// TIA Portal V18 program export: 1 tag tables, 0 data types, 3 data blocks, 8 code blocks (in call order from the OBs), 5 instance data blocks

VAR_GLOBAL   // PLC tag table "Default tag table"
   Tag_1 AT %M0.0 : Bool;
   System_Byte AT %MB1 : Byte;
   FirstScan AT %M1.0 : Bool;
   DiagStatusUpdate AT %M1.1 : Bool;
   AlwaysTRUE AT %M1.2 : Bool;
   AlwaysFALSE AT %M1.3 : Bool;
   Clock_Byte AT %MB0 : Byte;
   Clock_10Hz AT %M0.0 : Bool;
   Clock_5Hz AT %M0.1 : Bool;
   "Clock_2.5Hz" AT %M0.2 : Bool;
   Clock_2Hz AT %M0.3 : Bool;
   "Clock_1.25Hz" AT %M0.4 : Bool;
   Clock_1Hz AT %M0.5 : Bool;
   "Clock_0.625Hz" AT %M0.6 : Bool;
   "Clock_0.5Hz" AT %M0.7 : Bool;
   Tag_2 AT %M10.0 : Bool;
   Tag_3 AT %MW20 : Word;
   Tag_4 AT %M20.1 : Bool;
   Tag_5 AT %MD20 : Real;
   Tag_6 AT %M10.7 : Bool;
   Tag_7 AT %MD30 : DWord;
   Tag_8 AT %M10.5 : Bool;
END_VAR

DATA_BLOCK "DATA"   // DB2
{ S7_Optimized_Access := 'TRUE' }
VERSION : 0.1
// stored: AutoNumber true, DBAccessibleFromOPCUA true, DBAccessibleFromWebserver true, IsOnlyStoredInLoadMemory false, IsRetainMemResEnabled false, IsWriteProtectedInAS false, MemoryReserve 100
   VAR
      Str : String := '0+252+65526+5000+955+54+100+566';
      Str_1 : String[4];
      Val_1 : DInt;
      Val_2 : DInt;
      Val_3 : DInt;
   END_VAR
BEGIN
END_DATA_BLOCK

DATA_BLOCK "DB_CLOUD"   // DB1201
{ S7_Optimized_Access := 'FALSE' }
VERSION : 0.1
// stored: AutoNumber false, DBAccessibleFromOPCUA true, DBAccessibleFromWebserver true, IsOnlyStoredInLoadMemory false, IsWriteProtectedInAS false
   VAR
      P1S1O2 : Real := 1.0;
      P1S1CO2 : Real := 2.0;
      P1S1MT : Real := 3.0;
      P1S1H : Real := 4.0;
      P1S1PH : Real := 5.0;
      P1S2O2 : Real := 1.0;
      P1S2CO2 : Real := 2.0;
      P1S2MT : Real := 3.0;
      P1S2H : Real := 4.0;
      P1S2PH : Real := 5.0;
      P1S3O2 : Real := 1.0;
      P1S3CO2 : Real := 2.0;
      P1S3MT : Real := 3.0;
      P1S3H : Real := 4.0;
      P1S3PH : Real := 5.0;
      P2S1O2 : Real := 1.0;
      P2S1CO2 : Real := 2.0;
      P2S1MT : Real := 3.0;
      P2S1H : Real := 4.0;
      P2S1PH : Real := 5.0;
      P2S2O2 : Real := 1.0;
      P2S2CO2 : Real := 2.0;
      P2S2MT : Real := 3.0;
      P2S2H : Real := 4.0;
      P2S2PH : Real := 5.0;
      P2S3O2 : Real := 1.0;
      P2S3CO2 : Real := 2.0;
      P2S3MT : Real := 3.0;
      P2S3H : Real := 4.0;
      P2S3PH : Real := 5.0;
      P3S1O2 : Real := 1.0;
      P3S1CO2 : Real := 2.0;
      P3S1MT : Real := 3.0;
      P3S1H : Real := 4.0;
      P3S1PH : Real := 5.0;
      P3S2O2 : Real := 1.0;
      P3S2CO2 : Real := 2.0;
      P3S2MT : Real := 3.0;
      P3S2H : Real := 4.0;
      P3S2PH : Real := 5.0;
      P3S3O2 : Real := 1.0;
      P3S3CO2 : Real := 2.0;
      P3S3MT : Real := 3.0;
      P3S3H : Real := 4.0;
      P3S3PH : Real := 5.0;
      P4S1O2 : Real := 1.0;
      P4S1CO2 : Real := 2.0;
      P4S1MT : Real := 3.0;
      P4S1H : Real := 4.0;
      P4S1PH : Real := 5.0;
      P4S2O2 : Real := 1.0;
      P4S2CO2 : Real := 2.0;
      P4S2MT : Real := 3.0;
      P4S2H : Real := 4.0;
      P4S2PH : Real := 5.0;
      P4S3O2 : Real := 1.0;
      P4S3CO2 : Real := 2.0;
      P4S3MT : Real := 3.0;
      P4S3H : Real := 4.0;
      P4S3PH : Real := 5.0;
      P5S1O2 : Real := 1.0;
      P5S1CO2 : Real := 2.0;
      P5S1MT : Real := 3.0;
      P5S1H : Real := 4.0;
      P5S1PH : Real := 5.0;
      P5S2O2 : Real := 1.0;
      P5S2CO2 : Real := 2.0;
      P5S2MT : Real := 3.0;
      P5S2H : Real := 4.0;
      P5S2PH : Real := 5.0;
      P5S3O2 : Real := 1.0;
      P5S3CO2 : Real := 2.0;
      P5S3MT : Real := 3.0;
      P5S3H : Real := 4.0;
      P5S3PH : Real := 5.0;
      P6S1O2 : Real := 1.0;
      P6S1CO2 : Real := 2.0;
      P6S1MT : Real := 3.0;
      P6S1H : Real := 4.0;
      P6S1PH : Real := 5.0;
      P6S2O2 : Real := 1.0;
      P6S2CO2 : Real := 2.0;
      P6S2MT : Real := 3.0;
      P6S2H : Real := 4.0;
      P6S2PH : Real := 5.0;
      P6S3O2 : Real := 1.0;
      P6S3CO2 : Real := 2.0;
      P6S3MT : Real := 3.0;
      P6S3H : Real := 4.0;
      P6S3PH : Real := 5.0;
   END_VAR
BEGIN
END_DATA_BLOCK

DATA_BLOCK "DB_CLOUD_Simulation"   // DB1200
{ S7_Optimized_Access := 'FALSE' }
VERSION : 0.1
// stored: AutoNumber false, DBAccessibleFromOPCUA true, DBAccessibleFromWebserver true, IsOnlyStoredInLoadMemory false, IsWriteProtectedInAS false
   VAR RETAIN
      Array_1 : Array[1..90] of Real;
      P1S1CO2 : Real := 0.0;
      P1S1MT : Real := 1.0;
      P1S1H : Real := 2.0;
      P1S1PH : Real := 3.0;
      P1S2O2 : Real := 4.0;
      P1S2CO2 : Real := 5.0;
      P1S2MT : Real := 6.0;
      P1S2H : Real := 7.0;
      P1S2PH : Real := 8.0;
      P1S3O2 : Real := 9.0;
      P1S3CO2 : Real := 10.0;
      P1S3MT : Real := 11.0;
      P1S3H : Real := 12.0;
      P1S3PH : Real := 13.0;
      P2S1O2 : Real := 14.0;
      P2S1CO2 : Real := 15.0;
      P2S1MT : Real := 16.0;
      P2S1H : Real := 17.0;
      P2S1PH : Real := 18.0;
      P2S2O2 : Real := 19.0;
      P2S2CO2 : Real := 20.0;
      P2S2MT : Real := 21.0;
      P2S2H : Real := 22.0;
      P2S2PH : Real := 23.0;
      P2S3O2 : Real := 24.0;
      P2S3CO2 : Real := 25.0;
      P2S3MT : Real := 26.0;
      P2S3H : Real := 27.0;
      P2S3PH : Real := 28.0;
      P3S1O2 : Real := 29.0;
      P3S1CO2 : Real := 30.0;
      P3S1MT : Real := 31.0;
      P3S1H : Real := 32.0;
      P3S1PH : Real := 33.0;
      P3S2O2 : Real := 34.0;
      P3S2CO2 : Real := 35.0;
      P3S2MT : Real := 36.0;
      P3S2H : Real := 37.0;
      P3S2PH : Real := 38.0;
      P3S3O2 : Real := 39.0;
      P3S3CO2 : Real := 40.0;
      P3S3MT : Real := 41.0;
      P3S3H : Real := 42.0;
      P3S3PH : Real := 43.0;
      P4S1O2 : Real := 44.0;
      P4S1CO2 : Real := 45.0;
      P4S1MT : Real := 46.0;
      P4S1H : Real := 47.0;
      P4S1PH : Real := 48.0;
      P4S2O2 : Real := 49.0;
      P4S2CO2 : Real := 50.0;
      P4S2MT : Real := 51.0;
      P4S2H : Real := 52.0;
      P4S2PH : Real := 53.0;
      P4S3O2 : Real := 54.0;
      P4S3CO2 : Real := 55.0;
      P4S3MT : Real := 56.0;
      P4S3H : Real := 57.0;
      P4S3PH : Real := 58.0;
      P5S1O2 : Real := 59.0;
      P5S1CO2 : Real := 60.0;
      P5S1MT : Real := 61.0;
      P5S1H : Real := 62.0;
      P5S1PH : Real := 63.0;
      P5S2O2 : Real := 64.0;
      P5S2CO2 : Real := 65.0;
      P5S2MT : Real := 66.0;
      P5S2H : Real := 67.0;
      P5S2PH : Real := 68.0;
      P5S3O2 : Real := 69.0;
      P5S3CO2 : Real := 70.0;
      P5S3MT : Real := 71.0;
      P5S3H : Real := 72.0;
      P5S3PH : Real := 73.0;
      P6S1O2 : Real := 74.0;
      P6S1CO2 : Real := 75.0;
      P6S1MT : Real := 76.0;
      P6S1H : Real := 77.0;
      P6S1PH : Real := 78.0;
      P6S2O2 : Real := 79.0;
      P6S2CO2 : Real := 80.0;
      P6S2MT : Real := 81.0;
      P6S2H : Real := 82.0;
      P6S2PH : Real := 83.0;
      P6S3O2 : Real := 84.0;
      P6S3CO2 : Real := 85.0;
      P6S3MT : Real := 86.0;
      P6S3H : Real := 87.0;
      P6S3PH : Real := 88.0;
   END_VAR
BEGIN
   Array_1[1] := 0.0;
   Array_1[2] := 1.0;
   Array_1[3] := 2.0;
   Array_1[4] := 3.0;
   Array_1[5] := 4.0;
   Array_1[6] := 5.0;
   Array_1[7] := 6.0;
   Array_1[8] := 7.0;
   Array_1[9] := 8.0;
   Array_1[10] := 9.0;
   Array_1[11] := 10.0;
   Array_1[12] := 11.0;
   Array_1[13] := 12.0;
   Array_1[14] := 13.0;
   Array_1[15] := 14.0;
   Array_1[16] := 15.0;
   Array_1[17] := 16.0;
   Array_1[18] := 17.0;
   Array_1[19] := 18.0;
   Array_1[20] := 19.0;
   Array_1[21] := 20.0;
   Array_1[22] := 21.0;
   Array_1[23] := 22.0;
   Array_1[24] := 23.0;
   Array_1[25] := 24.0;
   Array_1[26] := 25.0;
   Array_1[27] := 26.0;
   Array_1[28] := 27.0;
   Array_1[29] := 28.0;
   Array_1[30] := 29.0;
   Array_1[31] := 30.0;
   Array_1[32] := 31.0;
   Array_1[33] := 32.0;
   Array_1[34] := 33.0;
   Array_1[35] := 34.0;
   Array_1[36] := 35.0;
   Array_1[37] := 36.0;
   Array_1[38] := 37.0;
   Array_1[39] := 38.0;
   Array_1[40] := 39.0;
   Array_1[41] := 40.0;
   Array_1[42] := 41.0;
   Array_1[43] := 42.0;
   Array_1[44] := 43.0;
   Array_1[45] := 44.0;
   Array_1[46] := 45.0;
   Array_1[47] := 46.0;
   Array_1[48] := 47.0;
   Array_1[49] := 48.0;
   Array_1[50] := 49.0;
   Array_1[51] := 50.0;
   Array_1[52] := 51.0;
   Array_1[53] := 52.0;
   Array_1[54] := 53.0;
   Array_1[55] := 54.0;
   Array_1[56] := 55.0;
   Array_1[57] := 56.0;
   Array_1[58] := 57.0;
   Array_1[59] := 58.0;
   Array_1[60] := 59.0;
   Array_1[61] := 60.0;
   Array_1[62] := 61.0;
   Array_1[63] := 62.0;
   Array_1[64] := 63.0;
   Array_1[65] := 64.0;
   Array_1[66] := 65.0;
   Array_1[67] := 66.0;
   Array_1[68] := 67.0;
   Array_1[69] := 68.0;
   Array_1[70] := 69.0;
   Array_1[71] := 70.0;
   Array_1[72] := 71.0;
   Array_1[73] := 72.0;
   Array_1[74] := 73.0;
   Array_1[75] := 74.0;
   Array_1[76] := 75.0;
   Array_1[77] := 76.0;
   Array_1[78] := 77.0;
   Array_1[79] := 78.0;
   Array_1[80] := 79.0;
   Array_1[81] := 80.0;
   Array_1[82] := 81.0;
   Array_1[83] := 82.0;
   Array_1[84] := 83.0;
   Array_1[85] := 84.0;
   Array_1[86] := 85.0;
   Array_1[87] := 86.0;
   Array_1[88] := 87.0;
   Array_1[89] := 88.0;
   Array_1[90] := 89.0;
END_DATA_BLOCK

ORGANIZATION_BLOCK "Main"   // OB1, LAD, ProgramCycle
TITLE = "Main Program Sweep (Cycle)"
{ S7_Optimized_Access := 'TRUE' }
VERSION : 0.1
// stored: AutoNumber true, IsIECCheckEnabled false, SetENOAutomatically false
   VAR_INPUT
      Initial_Call : Bool;   // Initial call of this OB
      Remanence : Bool;   // =True, if remanent data are available
   END_VAR
BEGIN

REGION Network 1
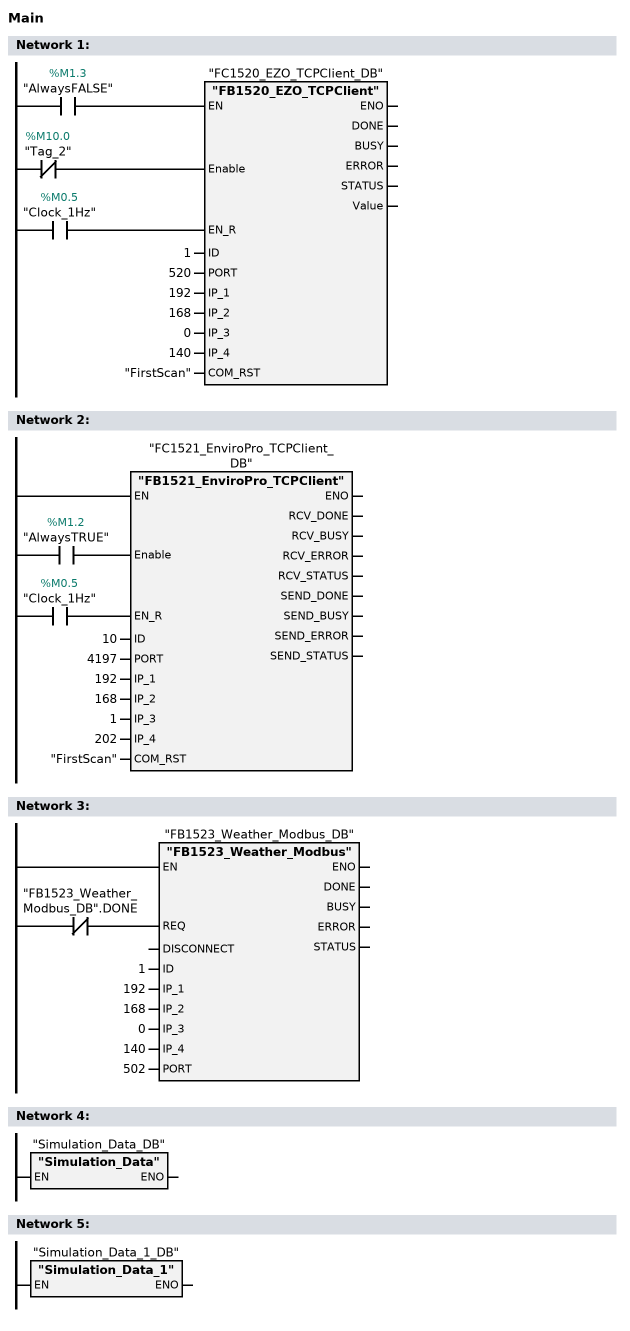
   RUNG wire#powerrail
      Contact( "AlwaysFALSE" )
      "FC1520_EZO_TCPClient_DB"(Enable := wire#w1, EN_R := wire#w2, ID := 1, PORT := 520, IP_1 := 192, IP_2 := 168, IP_3 := 0, IP_4 := 140, COM_RST := "FirstScan", DONE =>, BUSY =>, ERROR =>, STATUS =>, Value =>)
   END_RUNG
   RUNG wire#powerrail
      I_Contact( "Tag_2" )
   END_RUNG wire#w1
   RUNG wire#powerrail
      Contact( "Clock_1Hz" )
   END_RUNG wire#w2
   // the same network as SCL:
   IF "AlwaysFALSE" THEN
       "FC1520_EZO_TCPClient_DB"(Enable := NOT "Tag_2",   // "FB1520_EZO_TCPClient"
                               EN_R := "Clock_1Hz",
                               ID := 1,
                               PORT := 520,
                               IP_1 := 192,
                               IP_2 := 168,
                               IP_3 := 0,
                               IP_4 := 140,
                               COM_RST := "FirstScan");
   END_IF;
END_REGION

REGION Network 2
   RUNG wire#powerrail
      "FC1521_EnviroPro_TCPClient_DB"(Enable := wire#w1, EN_R := wire#w2, ID := 10, PORT := 4197, IP_1 := 192, IP_2 := 168, IP_3 := 1, IP_4 := 202, COM_RST := "FirstScan", RCV_DONE =>, RCV_BUSY =>, RCV_ERROR =>, RCV_STATUS =>, SEND_DONE =>, SEND_BUSY =>, SEND_ERROR =>, SEND_STATUS =>)
   END_RUNG
   RUNG wire#powerrail
      Contact( "AlwaysTRUE" )
   END_RUNG wire#w1
   RUNG wire#powerrail
      Contact( "Clock_1Hz" )
   END_RUNG wire#w2
   // the same network as SCL:
   "FC1521_EnviroPro_TCPClient_DB"(Enable := "AlwaysTRUE",   // "FB1521_EnviroPro_TCPClient"
                           EN_R := "Clock_1Hz",
                           ID := 10,
                           PORT := 4197,
                           IP_1 := 192,
                           IP_2 := 168,
                           IP_3 := 1,
                           IP_4 := 202,
                           COM_RST := "FirstScan");
END_REGION

REGION Network 3
   RUNG wire#powerrail
      "FB1523_Weather_Modbus_DB"(REQ := wire#w1, DISCONNECT :=, ID := 1, IP_1 := 192, IP_2 := 168, IP_3 := 0, IP_4 := 140, PORT := 502, DONE =>, BUSY =>, ERROR =>, STATUS =>)
   END_RUNG
   RUNG wire#powerrail
      I_Contact( "FB1523_Weather_Modbus_DB".DONE )
   END_RUNG wire#w1
   // the same network as SCL:
   "FB1523_Weather_Modbus_DB"(REQ := NOT "FB1523_Weather_Modbus_DB".DONE,   // "FB1523_Weather_Modbus"
                           ID := 1,
                           IP_1 := 192,
                           IP_2 := 168,
                           IP_3 := 0,
                           IP_4 := 140,
                           PORT := 502);
END_REGION

REGION Network 4
   RUNG wire#powerrail
      "Simulation_Data_DB"()
   END_RUNG
   // the same network as SCL:
   "Simulation_Data_DB"();   // "Simulation_Data"
END_REGION

REGION Network 5
   RUNG wire#powerrail
      "Simulation_Data_1_DB"()
   END_RUNG
   // the same network as SCL:
   "Simulation_Data_1_DB"();   // "Simulation_Data_1"
END_REGION
END_ORGANIZATION_BLOCK

FUNCTION_BLOCK "FB1520_EZO_TCPClient"
{ S7_Optimized_Access := 'TRUE' }
VERSION : 0.1
   VAR_INPUT 
      Enable : Bool;
      EN_R : Bool;
      ID : CONN_OUC := 16#0001;
      PORT : UInt := 4196;
      IP_1 : Byte := 192;
      IP_2 : Byte := 168;
      IP_3 : Byte := 1;
      IP_4 : Byte := 200;
   END_VAR

   VAR_OUTPUT 
      DONE : Bool;
      BUSY : Bool;
      ERROR : Bool;
      STATUS : Word;
      Value : Real;
   END_VAR

   VAR_IN_OUT 
      COM_RST : Bool;
   END_VAR

   VAR 
      CONNECT {InstructionName := 'TCON_IP_v4'; LibVersion := '1.0'; S7_SetPoint := 'False'} : TCON_IP_v4 := (64, 16#0001, (), TRUE, ([()]), (), ());
      RCV_DATA : Array[0..8] of Char;
      Done_Old : Bool;
      Pos_R : Int;
      TRCV_C1 {InstructionName := 'TRCV_C'; LibVersion := '3.2'; S7_SetPoint := 'False'} : TRCV_C;
      QT1 { S7_SetPoint := 'True'} : Bool;
      QT2 : Bool;
      T1 {InstructionName := 'TON_TIME'; LibVersion := '1.0'} : TON_TIME;
      T2 {InstructionName := 'TON_TIME'; LibVersion := '1.0'} : TON_TIME;
   END_VAR

   VAR_TEMP 
      ResetData : Array[0..8] of Char;
      RCV_Temp : Array[0..8] of Char;
      String_Temp_1 : String[9];
      String_Temp_2 : String[9];
   END_VAR


BEGIN
	
	REGION Initial
	    #CONNECT.ID := #ID;
	    #CONNECT.RemotePort := #PORT;
	    #CONNECT.RemoteAddress.ADDR[1] := #IP_1;
	    #CONNECT.RemoteAddress.ADDR[2] := #IP_2;
	    #CONNECT.RemoteAddress.ADDR[3] := #IP_3;
	    #CONNECT.RemoteAddress.ADDR[4] := #IP_4;
	    #TRCV_C1(EN_R := #EN_R,
	            CONT := #Enable,
	            LEN := 9,
	            ADHOC := TRUE,
	            DONE => #DONE,
	            BUSY => #BUSY,
	            ERROR => #ERROR,
	            STATUS => #STATUS,
	            CONNECT := #CONNECT,
	            DATA := #RCV_Temp,
	            COM_RST := #COM_RST);
	    
	END_REGION
	REGION Split Data
	    IF #TRCV_C1.DONE AND NOT #Done_Old THEN
	        #RCV_DATA := #RCV_Temp;
	        #RCV_Temp := #ResetData;
	    END_IF;
	    Chars_TO_Strg(Chars := #RCV_DATA,
	                  pChars := 0,
	                  Cnt := 0,
	                  Strg => #String_Temp_1);
	    #Pos_R := FIND(IN1 := #String_Temp_1, IN2 := '$R');
	    #String_Temp_2 := CONCAT_STRING(IN1 := '$R', IN2 := #String_Temp_1);
	    #Value := STRING_TO_REAL(MID_STRING(IN := #String_Temp_2, L := #Pos_R - 1, P := 2));
	    
	END_REGION
	REGION Restart Comunication
	    #T1(IN:= NOT #DONE AND NOT #QT2,
	       PT:=T#4s,
	       Q=>#QT1);
	   #T2(IN := #QT1,
	       PT := T#1s,
	       Q => #QT2);
	   #COM_RST := #QT1;
	   
	END_REGION
	
	#Done_Old := #TRCV_C1.DONE;
	
	
END_FUNCTION_BLOCK

FUNCTION_BLOCK "FB1521_EnviroPro_TCPClient"
{ S7_Optimized_Access := 'TRUE' }
VERSION : 0.1
   VAR_INPUT 
      Enable : Bool;
      EN_R : Bool;
      ID : CONN_OUC := 16#0001;
      PORT : UInt := 4196;
      IP_1 : Byte := 192;
      IP_2 : Byte := 168;
      IP_3 : Byte := 1;
      IP_4 : Byte := 200;
   END_VAR

   VAR_OUTPUT 
      RCV_DONE : Bool;
      RCV_BUSY : Bool;
      RCV_ERROR : Bool;
      RCV_STATUS : Word;
      SEND_DONE : Bool;
      SEND_BUSY : Bool;
      SEND_ERROR : Bool;
      SEND_STATUS : Word;
   END_VAR

   VAR_IN_OUT 
      COM_RST : Bool;
   END_VAR

   VAR 
      CONNECT {InstructionName := 'TCON_IP_v4'; LibVersion := '1.0'; S7_SetPoint := 'False'} : TCON_IP_v4 := (64, 16#0001, (), TRUE, ([()]), (), ());
      RCV_DATA : Array[1..90] of Char;
      RCV_VWC : Array[1..9] of Real;
      RCV_ECe : Array[1..9] of Real;
      RCV_TEMP : Array[1..9] of Real;
      Done_Old : Bool;
      Pos_R : Int;
      TRCV_C {InstructionName := 'TRCV_C'; LibVersion := '3.2'; S7_SetPoint := 'False'} : TRCV_C;
      TSEND_C {InstructionName := 'TSEND_C'; LibVersion := '3.2'} : TSEND_C;
      Send_Cmd : String[12] := '7C!<CR><LF>';
      Count_Cmd : Int;
      TON_1 {InstructionName := 'TON_TIME'; LibVersion := '1.0'} : TON_TIME;
      TON_2 {InstructionName := 'TON_TIME'; LibVersion := '1.0'} : TON_TIME;
      QT1 { ExternalAccessible := 'False'; ExternalVisible := 'False'; ExternalWritable := 'False'} : Bool;
      QT2 { ExternalAccessible := 'False'; ExternalVisible := 'False'; ExternalWritable := 'False'} : Bool;
   END_VAR

   VAR_TEMP 
      ResetData : Array[1..90] of Char;
      RCV_Temp1 : Array[1..90] of Char;
      Cmd_VWC : UInt;
      Cmd_ECe : UInt;
      Cmd_TEMP : UInt;
      Cmd_VWC_String : String[10];
      Cmd_ECe_String : String[10];
      Cmd_TEMP_String : String[10];
      String_Temp_1 : String[90];
      String_Temp_2 : String[90];
      String_Temp_3 : String[90];
   END_VAR


BEGIN
	REGION Initial
	    #CONNECT.ID := #ID;
	    #CONNECT.RemotePort := #PORT;
	    #CONNECT.RemoteAddress.ADDR[1] := #IP_1;
	    #CONNECT.RemoteAddress.ADDR[2] := #IP_2;
	    #CONNECT.RemoteAddress.ADDR[3] := #IP_3;
	    #CONNECT.RemoteAddress.ADDR[4] := #IP_4;
	    #TSEND_C(REQ:= #EN_R,
	             CONT:=#Enable,
	             LEN:=0,
	             DONE=>#SEND_DONE,
	             BUSY=>#SEND_BUSY,
	             ERROR=>#SEND_ERROR,
	             STATUS=>#SEND_STATUS,
	             CONNECT:=#CONNECT,
	             DATA:=#Send_Cmd,
	             COM_RST:=#COM_RST);
	    #TRCV_C(EN_R := #SEND_DONE,
	            CONT :=#Enable,
	            LEN := 80,
	            ADHOC := TRUE,
	            DONE => #RCV_DONE,
	            BUSY => #RCV_BUSY,
	            ERROR => #RCV_ERROR,
	            STATUS => #RCV_STATUS,
	            CONNECT := #CONNECT,
	            DATA := #RCV_Temp1,
	            COM_RST := #COM_RST);
	END_REGION
	
	REGION Split Data
	    IF #TRCV_C.DONE AND NOT #Done_Old THEN
	        #RCV_DATA := #RCV_Temp1;
	        #RCV_Temp1 := #ResetData;
	    END_IF;
	
	    //Read VWC 7C3!<CR><LF>
	    IF #Count_Cmd = 0 THEN
	        #Send_Cmd := '7C!<CR><LF>';
	        Chars_TO_Strg(Chars := #RCV_DATA,
	                      pChars := 0,
	                      Cnt := 0,
	                      Strg => #String_Temp_1);
	        Chars_TO_Strg(Chars := #RCV_DATA,
	                      pChars := 0,
	                      Cnt := 10,
	                      Strg => #Cmd_VWC_String);
	        #Cmd_VWC := STRING_TO_UINT(#Cmd_VWC_String);
	        IF #Cmd_VWC > 10 THEN
	            #Send_Cmd := '7D0!<CR><LF>';
	        END_IF;
	        IF (FIND(IN1 := #String_Temp_1, IN2 := '+') > 0) THEN
	            "FC1522_Split_EnviroPro"(In_String:=#String_Temp_1, RCV_DATA=>#RCV_VWC);
	            #RCV_DATA := #ResetData;
	            #Count_Cmd := 1;
	        END_IF;
	    END_IF;
	    //Read ECe
	    IF #Count_Cmd = 1 THEN
	        #Send_Cmd := '7C1!<CR><LF>';
	        Chars_TO_Strg(Chars := #RCV_DATA,
	                      pChars := 0,
	                      Cnt := 0,
	                      Strg => #String_Temp_2);
	        Chars_TO_Strg(Chars := #RCV_DATA,
	                      pChars := 0,
	                      Cnt := 10,
	                      Strg => #Cmd_ECe_String);
	        #Cmd_ECe := STRING_TO_UINT(#Cmd_ECe_String);
	        IF #Cmd_ECe > 10 THEN
	            #Send_Cmd := '7D0!<CR><LF>';
	        END_IF;
	        IF (FIND(IN1 := #String_Temp_2, IN2 := '+') > 0) THEN
	            "FC1522_Split_EnviroPro"(In_String := #String_Temp_2, RCV_DATA => #RCV_ECe);
	            #RCV_DATA := #ResetData;
	            #Count_Cmd := 2;
	        END_IF;
	    END_IF;
	    //Read TEMP
	    IF #Count_Cmd = 2 THEN
	        #Send_Cmd := '7C2!<CR><LF>';
	        Chars_TO_Strg(Chars := #RCV_DATA,
	                      pChars := 0,
	                      Cnt := 0,
	                      Strg => #String_Temp_3);
	        Chars_TO_Strg(Chars := #RCV_DATA,
	                      pChars := 0,
	                      Cnt := 10,
	                      Strg => #Cmd_TEMP_String);
	        #Cmd_TEMP := STRING_TO_UINT(#Cmd_TEMP_String);
	        IF #Cmd_TEMP > 10 THEN
	            #Send_Cmd := '7D0!<CR><LF>';
	        END_IF;
	        IF (FIND(IN1 := #String_Temp_3, IN2 := '+') > 0) THEN
	            "FC1522_Split_EnviroPro"(In_String := #String_Temp_3, RCV_DATA => #RCV_TEMP);
	           #RCV_DATA := #ResetData;
	            #Count_Cmd := 0;
	        END_IF;
	    END_IF;
	END_REGION
	
	#Done_Old := #TRCV_C.DONE;
	
	REGION Restart Comunication
	    #TON_1(IN := (NOT #SEND_DONE AND NOT #QT2),
	           PT := T#5s,
	           Q => #QT1);
	    #TON_2(IN := #QT1,
	           PT := T#1s,
	           Q => #QT2);
	    #COM_RST := #QT1;
	    IF #COM_RST THEN
	        #Count_Cmd := 0;
	    END_IF;
	    
	END_REGION
	
END_FUNCTION_BLOCK

FUNCTION "FC1522_Split_EnviroPro" : Void
{ S7_Optimized_Access := 'TRUE' }
VERSION : 0.1
   VAR_INPUT 
      In_String : String;
   END_VAR

   VAR_OUTPUT 
      RCV_DATA : Array[0..8] of Real;
   END_VAR

   VAR_TEMP 
      Cnt : UInt;
      String_Temp : String;
      i : Int;
      j : Int;
      k : Int;
      Char_temp : Array[1..92] of Char;
      Leng_1 : Int;
      Pos_1 : Array[0..9] of Int;
   END_VAR


BEGIN
	#String_Temp := CONCAT_STRING(IN1 := '+', IN2 := #In_String);
	#String_Temp := CONCAT_STRING(IN1 := #String_Temp, IN2 := '+');
	Strg_TO_Chars(Strg := #String_Temp,
	              pChars := 0,
	              Cnt => #Cnt,
	              Chars := #Char_temp);
	#Leng_1 := LEN(#String_Temp);
	FOR #i := 1 TO #Leng_1 DO
	    IF #Char_temp[#i] = '+' THEN
	        IF #j < 10 THEN (* Đảm bảo i không tràn *)
	            #Pos_1[#j] := #i;
	            #j := #j + 1;
	        END_IF;
	    END_IF;
	    
	END_FOR;
	FOR #k := 0 TO 8 DO
	    #RCV_DATA[#k] := STRING_TO_REAL(MID_STRING(IN := #In_String, L := #Pos_1[#k + 1] - #Pos_1[#k] - 1, P := #Pos_1[#k]));
	END_FOR;
	
	
	
END_FUNCTION

FUNCTION_BLOCK "FB1523_Weather_Modbus"
{ S7_Optimized_Access := 'TRUE' }
VERSION : 0.1
   VAR_INPUT 
      REQ : Bool;
      DISCONNECT : Bool;
      ID : CONN_OUC := 16#1;
      IP_1 : Byte := 192;
      IP_2 : Byte := 168;
      IP_3 : Byte := 0;
      IP_4 : Byte := 140;
      PORT : UInt := 502;
   END_VAR

   VAR_OUTPUT 
      DONE : Bool;
      BUSY : Bool;
      ERROR : Bool;
      STATUS : Word;
   END_VAR

   VAR 
      CONNECT {InstructionName := 'TCON_IP_v4'; LibVersion := '1.0'; S7_SetPoint := 'False'} : TCON_IP_v4 := (64, 16#1, (), True, ([()]), (), ());
      MB_CLIENT {InstructionName := 'MB_CLIENT'; LibVersion := '4.1'} : MB_CLIENT;
      RCV_DATA { S7_SetPoint := 'True'} : Array[0..13] of DInt;
   END_VAR


BEGIN
	REGION Initial
	    #CONNECT.ID := #ID;
	    #CONNECT.RemotePort := #PORT;
	    #CONNECT.RemoteAddress.ADDR[1] := #IP_1;
	    #CONNECT.RemoteAddress.ADDR[2] := #IP_2;
	    #CONNECT.RemoteAddress.ADDR[3] := #IP_3;
	    #CONNECT.RemoteAddress.ADDR[4] := #IP_4;
	    #MB_CLIENT(REQ:=#REQ,
	               DISCONNECT:=#DISCONNECT,
	               MB_MODE:=0,
	               MB_DATA_ADDR:=30001,
	               MB_DATA_LEN:=28,
	               DONE=>#DONE,
	               BUSY=>#BUSY,
	               ERROR=>#ERROR,
	               STATUS=>#STATUS,
	               MB_DATA_PTR:=#RCV_DATA,
	               CONNECT:=#CONNECT);
	    
	END_REGION
	
	
END_FUNCTION_BLOCK

FUNCTION_BLOCK "Simulation_Data"
{ S7_Optimized_Access := 'TRUE' }
VERSION : 0.1
   VAR 
      Old_Clock : Bool;
      i : Int;
   END_VAR


BEGIN
	IF "Clock_1Hz" AND NOT #Old_Clock THEN
	    "DB_CLOUD".P1S1O2 := "DB_CLOUD".P1S1O2 + 1.0;
	    "DB_CLOUD".P1S1CO2 := "DB_CLOUD".P1S1CO2 + 1.0;
	    "DB_CLOUD".P1S1MT := "DB_CLOUD".P1S1MT + 1.0;
	    "DB_CLOUD".P1S1H := "DB_CLOUD".P1S1H + 1.0;
	    "DB_CLOUD".P1S1PH := "DB_CLOUD".P1S1PH + 1.0;
	    
	    "DB_CLOUD".P1S2O2 := "DB_CLOUD".P1S2O2 + 1.0;
	    "DB_CLOUD".P1S2CO2 := "DB_CLOUD".P1S2CO2 + 1.0;
	    "DB_CLOUD".P1S2MT := "DB_CLOUD".P1S2MT + 1.0;
	    "DB_CLOUD".P1S2H := "DB_CLOUD".P1S2H + 1.0;
	    "DB_CLOUD".P1S2PH := "DB_CLOUD".P1S2PH + 1.0;
	    
	    "DB_CLOUD".P1S3O2 := "DB_CLOUD".P1S3O2 + 1.0;
	    "DB_CLOUD".P1S3CO2 := "DB_CLOUD".P1S3CO2 + 1.0;
	    "DB_CLOUD".P1S3MT := "DB_CLOUD".P1S3MT + 1.0;
	    "DB_CLOUD".P1S3H := "DB_CLOUD".P1S3H + 1.0;
	    "DB_CLOUD".P1S3PH := "DB_CLOUD".P1S3PH + 1.0;
	    //=======================================
	    "DB_CLOUD".P2S1O2 := "DB_CLOUD".P2S1O2 + 1.0;
	    "DB_CLOUD".P2S1CO2 := "DB_CLOUD".P2S1CO2 + 1.0;
	    "DB_CLOUD".P2S1MT := "DB_CLOUD".P2S1MT + 1.0;
	    "DB_CLOUD".P2S1H := "DB_CLOUD".P2S1H + 1.0;
	    "DB_CLOUD".P2S1PH := "DB_CLOUD".P2S1PH + 1.0;
	    
	    "DB_CLOUD".P2S2O2 := "DB_CLOUD".P2S2O2 + 1.0;
	    "DB_CLOUD".P2S2CO2 := "DB_CLOUD".P2S2CO2 + 1.0;
	    "DB_CLOUD".P2S2MT := "DB_CLOUD".P2S2MT + 1.0;
	    "DB_CLOUD".P2S2H := "DB_CLOUD".P2S2H + 1.0;
	    "DB_CLOUD".P2S2PH := "DB_CLOUD".P2S2PH + 1.0;
	    
	    "DB_CLOUD".P2S3O2 := "DB_CLOUD".P2S3O2 + 1.0;
	    "DB_CLOUD".P2S3CO2 := "DB_CLOUD".P2S3CO2 + 1.0;
	    "DB_CLOUD".P2S3MT := "DB_CLOUD".P2S3MT + 1.0;
	    "DB_CLOUD".P2S3H := "DB_CLOUD".P2S3H + 1.0;
	    "DB_CLOUD".P2S3PH := "DB_CLOUD".P2S3PH + 1.0;
	    //=======================================
	    "DB_CLOUD".P3S1O2 := "DB_CLOUD".P3S1O2 + 1.0;
	    "DB_CLOUD".P3S1CO2 := "DB_CLOUD".P3S1CO2 + 1.0;
	    "DB_CLOUD".P3S1MT := "DB_CLOUD".P3S1MT + 1.0;
	    "DB_CLOUD".P3S1H := "DB_CLOUD".P3S1H + 1.0;
	    "DB_CLOUD".P3S1PH := "DB_CLOUD".P3S1PH + 1.0;
	    
	    "DB_CLOUD".P3S2O2 := "DB_CLOUD".P3S2O2 + 1.0;
	    "DB_CLOUD".P3S2CO2 := "DB_CLOUD".P3S2CO2 + 1.0;
	    "DB_CLOUD".P3S2MT := "DB_CLOUD".P3S2MT + 1.0;
	    "DB_CLOUD".P3S2H := "DB_CLOUD".P3S2H + 1.0;
	    "DB_CLOUD".P3S2PH := "DB_CLOUD".P3S2PH + 1.0;
	    
	    "DB_CLOUD".P3S3O2 := "DB_CLOUD".P3S3O2 + 1.0;
	    "DB_CLOUD".P3S3CO2 := "DB_CLOUD".P3S3CO2 + 1.0;
	    "DB_CLOUD".P3S3MT := "DB_CLOUD".P3S3MT + 1.0;
	    "DB_CLOUD".P3S3H := "DB_CLOUD".P3S3H + 1.0;
	    "DB_CLOUD".P3S3PH := "DB_CLOUD".P3S3PH + 1.0;
	    //==========================
	    "DB_CLOUD".P4S1O2 := "DB_CLOUD".P4S1O2 + 1.0;
	    "DB_CLOUD".P4S1CO2 := "DB_CLOUD".P4S1CO2 + 1.0;
	    "DB_CLOUD".P4S1MT := "DB_CLOUD".P4S1MT + 1.0;
	    "DB_CLOUD".P4S1H := "DB_CLOUD".P4S1H + 1.0;
	    "DB_CLOUD".P4S1PH := "DB_CLOUD".P4S1PH + 1.0;
	    
	    "DB_CLOUD".P4S2O2 := "DB_CLOUD".P4S2O2 + 1.0;
	    "DB_CLOUD".P4S2CO2 := "DB_CLOUD".P4S2CO2 + 1.0;
	    "DB_CLOUD".P4S2MT := "DB_CLOUD".P4S2MT + 1.0;
	    "DB_CLOUD".P4S2H := "DB_CLOUD".P4S2H + 1.0;
	    "DB_CLOUD".P4S2PH := "DB_CLOUD".P4S2PH + 1.0;
	    
	    "DB_CLOUD".P4S3O2 := "DB_CLOUD".P4S3O2 + 1.0;
	    "DB_CLOUD".P4S3CO2 := "DB_CLOUD".P4S3CO2 + 1.0;
	    "DB_CLOUD".P4S3MT := "DB_CLOUD".P4S3MT + 1.0;
	    "DB_CLOUD".P4S3H := "DB_CLOUD".P4S3H + 1.0;
	    "DB_CLOUD".P4S3PH := "DB_CLOUD".P4S3PH + 1.0;
	    //==================================
	    "DB_CLOUD".P5S1O2 := "DB_CLOUD".P5S1O2 + 1.0;
	    "DB_CLOUD".P5S1CO2 := "DB_CLOUD".P5S1CO2 + 1.0;
	    "DB_CLOUD".P5S1MT := "DB_CLOUD".P5S1MT + 1.0;
	    "DB_CLOUD".P5S1H := "DB_CLOUD".P5S1H + 1.0;
	    "DB_CLOUD".P5S1PH := "DB_CLOUD".P5S1PH + 1.0;
	    
	    "DB_CLOUD".P5S2O2 := "DB_CLOUD".P5S2O2 + 1.0;
	    "DB_CLOUD".P5S2CO2 := "DB_CLOUD".P5S2CO2 + 1.0;
	    "DB_CLOUD".P5S2MT := "DB_CLOUD".P5S2MT + 1.0;
	    "DB_CLOUD".P5S2H := "DB_CLOUD".P5S2H + 1.0;
	    "DB_CLOUD".P5S2PH := "DB_CLOUD".P5S2PH + 1.0;
	    
	    "DB_CLOUD".P5S3O2 := "DB_CLOUD".P5S3O2 + 1.0;
	    "DB_CLOUD".P5S3CO2 := "DB_CLOUD".P5S3CO2 + 1.0;
	    "DB_CLOUD".P5S3MT := "DB_CLOUD".P5S3MT + 1.0;
	    "DB_CLOUD".P5S3H := "DB_CLOUD".P5S3H + 1.0;
	    "DB_CLOUD".P5S3PH := "DB_CLOUD".P5S3PH + 1.0;
	    //==============================
	    "DB_CLOUD".P6S1O2 := "DB_CLOUD".P6S1O2 + 1.0;
	    "DB_CLOUD".P6S1CO2 := "DB_CLOUD".P6S1CO2 + 1.0;
	    "DB_CLOUD".P6S1MT := "DB_CLOUD".P6S1MT + 1.0;
	    "DB_CLOUD".P6S1H := "DB_CLOUD".P6S1H + 1.0;
	    "DB_CLOUD".P6S1PH := "DB_CLOUD".P6S1PH + 1.0;
	    
	    "DB_CLOUD".P6S2O2 := "DB_CLOUD".P6S2O2 + 1.0;
	    "DB_CLOUD".P6S2CO2 := "DB_CLOUD".P6S2CO2 + 1.0;
	    "DB_CLOUD".P6S2MT := "DB_CLOUD".P6S2MT + 1.0;
	    "DB_CLOUD".P6S2H := "DB_CLOUD".P6S2H + 1.0;
	    "DB_CLOUD".P6S2PH := "DB_CLOUD".P6S2PH + 1.0;
	    
	    "DB_CLOUD".P6S3O2 := "DB_CLOUD".P6S3O2 + 1.0;
	    "DB_CLOUD".P6S3CO2 := "DB_CLOUD".P6S3CO2 + 1.0;
	    "DB_CLOUD".P6S3MT := "DB_CLOUD".P6S3MT + 1.0;
	    "DB_CLOUD".P6S3H := "DB_CLOUD".P6S3H + 1.0;
	    "DB_CLOUD".P6S3PH := "DB_CLOUD".P6S3PH + 1.0;
	   
	  
	END_IF;
	#Old_Clock := "Clock_1Hz";
END_FUNCTION_BLOCK

FUNCTION_BLOCK "Simulation_Data_1"
{ S7_Optimized_Access := 'TRUE' }
VERSION : 0.1
   VAR 
      Old_Clock : Bool;
      i : Int;
   END_VAR


BEGIN
	IF "Clock_1Hz" AND NOT #Old_Clock THEN
	    FOR #i := 1 TO 90 DO
	        "DB_CLOUD_Simulation".Array_1[#i] := "DB_CLOUD_Simulation".Array_1[#i] + 1;
	        IF "DB_CLOUD_Simulation".Array_1[#i] > 600 THEN
	            "DB_CLOUD_Simulation".Array_1[#i] := 0;
	        END_IF;
	    END_FOR;
	   
	    
	    
	    
	END_IF;
	#Old_Clock := "Clock_1Hz";
END_FUNCTION_BLOCK

FUNCTION "StringToReal" : Void
{ S7_Optimized_Access := 'TRUE' }
VERSION : 0.1
   VAR_INPUT 
      In : String;
   END_VAR

   VAR_OUTPUT 
      Out : Real;
   END_VAR


BEGIN
	#Out := STRING_TO_REAL(#In);
END_FUNCTION

DATA_BLOCK "FB1523_Weather_Modbus_DB"   // DB8
VERSION : 0.1
// stored: AutoNumber true, DBAccessibleFromOPCUA true, DBAccessibleFromWebserver true, InstanceOfName FB1523_Weather_Modbus, InstanceOfType FB
"FB1523_Weather_Modbus"
BEGIN
END_DATA_BLOCK

DATA_BLOCK "FC1520_EZO_TCPClient_DB"   // DB6
VERSION : 0.1
// stored: AutoNumber true, DBAccessibleFromOPCUA true, DBAccessibleFromWebserver true, InstanceOfName FB1520_EZO_TCPClient, InstanceOfType FB
"FB1520_EZO_TCPClient"
BEGIN
END_DATA_BLOCK

DATA_BLOCK "FC1521_EnviroPro_TCPClient_DB"   // DB4
VERSION : 0.1
// stored: AutoNumber true, DBAccessibleFromOPCUA true, DBAccessibleFromWebserver true, InstanceOfName FB1521_EnviroPro_TCPClient, InstanceOfType FB
"FB1521_EnviroPro_TCPClient"
BEGIN
END_DATA_BLOCK

DATA_BLOCK "Simulation_Data_1_DB"   // DB3
VERSION : 0.1
// stored: AutoNumber true, DBAccessibleFromOPCUA true, DBAccessibleFromWebserver true, InstanceOfName Simulation_Data_1, InstanceOfType FB
"Simulation_Data_1"
BEGIN
END_DATA_BLOCK

DATA_BLOCK "Simulation_Data_DB"   // DB1
VERSION : 0.1
// stored: AutoNumber true, DBAccessibleFromOPCUA true, DBAccessibleFromWebserver true, InstanceOfName Simulation_Data, InstanceOfType FB
"Simulation_Data"
BEGIN
END_DATA_BLOCK
